{attribute 'qualified_only'}
{attribute 'strict'}
TYPE StandardPlane :
(
	XY := Tc2_PlcInterpolation.E_NciGeoPlane.E_NciGeoPlaneXY,
	ZX := Tc2_PlcInterpolation.E_NciGeoPlane.E_NciGeoPlaneZX,
	YZ := Tc2_PlcInterpolation.E_NciGeoPlane.E_NciGeoPlaneYZ
) INT;
END_TYPE

(* stored: Version 1.1.0.1, ProductVersion 3.1.4024.12
   DUT StandardPlane: Id {3a0413c6-4c14-45a3-a32a-40bbee1cc24e} *)
